PROGRAM P_Inputs
VAR
	fbNormPa :  FB_Normalize;
	fbNormPb :  FB_Normalize;
	fbNormPs :  FB_Normalize;
	fbNormPaLower : FB_Normalize;
	
	fbNormPistonPosition : FB_PositionInputScaling;
	fbNormSpoolPosition : FB_JoystickInputScaling;
	fbJoystick : FB_JoystickInputScaling;
	fbFlow	: FB_JoystickInputScaling;

	fPa : LREAL;
	fPb : LREAL;
	fPs : LREAL;
	fPaLower : LREAL;
	
	fPistonPosition : LREAL;
END_VAR

fbNormPa(
	nRawInput := G_Inputs.nRawPa,
	fMaxValue := 400.0, 			// [Bar]
	fNormalizedInput => G_OPC.fPa
);

fbNormPb(
	nRawInput := G_Inputs.nRawPb,
	fMaxValue := 400.0, 			// [Bar]
	fNormalizedInput => G_OPC.fPb
);

fbNormPs(
	nRawInput := G_Inputs.nRawPs,
	fMaxValue := 400.0, 			// [Bar]
	fNormalizedInput => G_OPC.fPs
);

fbNormPistonPosition(
	nRawInput := G_Inputs.nRawPistonPosition,
	
	fMaxInputValue := 16090.0,
	fMinInputValue := 125.0,
	fMaxOutputValue := 0.5,
	fMinOutputValue := 0.0,	
	
	fOutput => G_OPC.fPistonPosMeasured,
	fActual => G_OPC.fPistonPosition
);
	
fbJoystick(
	nRawInput := G_Inputs.nRawJoystick,
	fMaxValue := 1.0,
	bEnable := (G_Mode.bRunning AND G_Mode.bManual),
	
	fMaxInputValue := 14746.0,
	fMinInputValue := 1617.0,
	fNeutralInputValue := 8160.0,
	fNeutralDeadband := 100.0,
	
	fOutput => G_OPC.fJoystick
);

fbNormPaLower(
	nRawInput := G_Inputs.nRawPaLower,
	fMaxValue := 400.0, 			// [Bar]
	fNormalizedInput => G_OPC.fPaLower
);

fbNormSpoolPosition(
	nRawInput := G_Inputs.nRawSpoolPosition,
	fMaxValue := 1.0,
	bEnable := TRUE,
	
	fNeutralInputValue := 8355.0,
	fMaxInputValue := 12645.0,
	fMinInputValue := 4071,
	fNeutralDeadband := 15.0,
	
	fOutput => G_OPC.fSpoolPosition
);

fbFlow(
	bEnable := TRUE,
	nRawInput := G_Inputs.nRawFlowSensor,
	fMaxValue := 150.0, // [l/min]
	
	fMaxInputValue := 32767.0,
	fMinInputValue := 0,
	fNeutralInputValue := 15270.0,
	fNeutralDeadband := 25.0,
	
	fOutput => G_OPC.fFlow
);

END_PROGRAM

(* stored: Version 1.1.0.1, ProductVersion 3.1.4024.12
   POU P_Inputs: Id {94ed4cce-6a16-4a20-9eff-b4a1e6338584}, SpecialFunc None *)
